FUNCTION JoinStrings : STRING
VAR_INPUT
	str1, str2, separator : STRING;
END_VAR
VAR
END_VAR

JoinStrings := CONCAT(str1, separator);
JoinStrings := CONCAT(JoinStrings, str2);

END_FUNCTION

(* stored: Version 1.1.0.1, ProductVersion 3.1.4024.11
   POU JoinStrings: Id {b1a99a54-d937-4f0f-910c-7d8c766642fe}, SpecialFunc None *)
